{attribute addProperty BoxType "EL3164-0000-0020"}
{attribute addProperty Id "StatusAT %I*Status_EBD4BD798ValueAT %I*INT2"}
{attribute addProperty CRC "3184610221"}
{attribute addProperty SizeInBites "80"}
{attribute addProperty SizeInBytes "10"}
TYPE AI_Standard_Channel_BDD14BAD :
STRUCT
	{attribute addProperty Name "Status"}
	Status AT %I* : Status_EBD4BD79;
	{attribute addProperty Name "Value"}
	Value AT %I* : INT;
END_STRUCT
END_TYPE

(* stored: Version 1.2.0.0, ProductVersion 3.1.4024.9
   DUT AI_Standard_Channel_BDD14BAD: Id {1cede855-2aa7-48cc-9734-74a6b422f7a7} *)
